PROGRAM MAIN
VAR
	bStart : BOOL;
	fbCsv : FB_CsvFileWriter;
	iFileWriter : I_FileWriter;
	sMessage : STRING := 'This is third message in the file';
END_VAR

iFileWriter := fbCsv;

IF bStart THEN
	iFileWriter.WriteEvent(sMessage);
	bStart := FALSE;
END_IF
fbCsv();

END_PROGRAM

(* stored: Version 1.1.0.1, ProductVersion 3.1.4024.16
   POU MAIN: Id {a3d65056-a026-4064-93e5-092b5fb5e321}, SpecialFunc None *)
